TYPE defSCARATasks :
STRUCT
END_STRUCT
END_TYPE

(* stored: Version 1.1.0.1, ProductVersion 3.1.4024.0
   DUT defSCARATasks: Id {a55cbc21-dfa7-4f6a-ba02-57fa5e05d7a1} *)
